// TIA Portal V17 export
// export: Created 2024-08-07T21:44:10.1007869Z, ExportSetting WithDefaults, DisplayName Totally Integrated Automation Portal, DisplayVersion V17 Update 7, DisplayName TIA Portal Openness, DisplayVersion V17 Update 7, DisplayName TIA Portal Version Control Interface, DisplayVersion V17, DisplayName SINAMICS Startdrive Advanced, DisplayVersion V17 SP2, DisplayName SINAMICS Startdrive G110M, G120, G120C, G120D, G120P, G115D, DisplayVersion V17 SP2, DisplayName SINAMICS Startdrive G130, G150, S120, S150, SINAMICS MV, S210, DisplayVersion V17 SP2, DisplayName STEP 7 Professional, DisplayVersion V17 Update 7, DisplayName STEP 7 Safety, DisplayVersion V17 Update 6, DisplayName WinCC Advanced / Unified PC, DisplayVersion V17 Update 7
FUNCTION "FC_DMC" : Void   // FC2012, LAD
{ S7_Optimized_Access := 'TRUE' }
VERSION : 0.1
// stored: AutoNumber false, IsIECCheckEnabled false, SetENOAutomatically false, UDAEnableTagReadback false
   VAR_TEMP
      stationName1 : WString;
      stationName2 : WString;
   END_VAR
BEGIN

REGION Network 1: SET DMC CONNECTION BLOCK
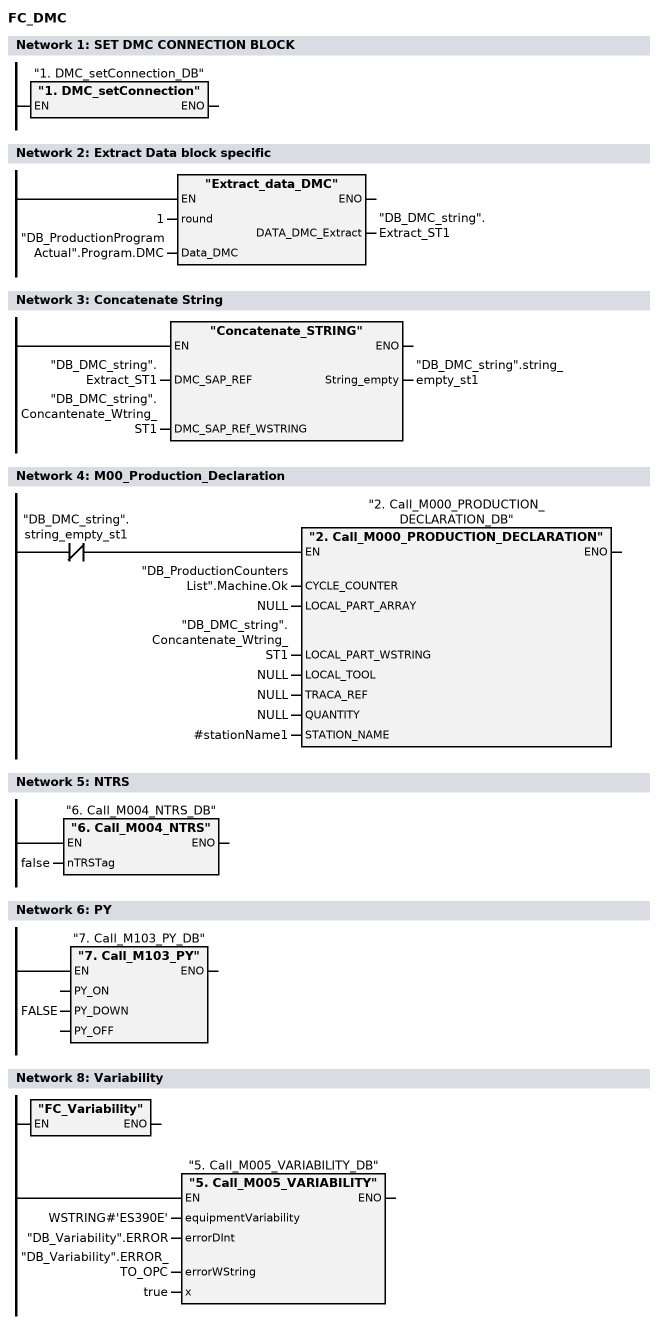
   RUNG wire#powerrail
      "1. DMC_setConnection_DB"()
   END_RUNG
   // the same network as SCL:
   "1. DMC_setConnection_DB"();   // "1. DMC_setConnection"
END_REGION

REGION Network 2: Extract Data block specific
   RUNG wire#powerrail
      "Extract_data_DMC"(round := 1, Data_DMC := "DB_ProductionProgramActual".Program.DMC, DATA_DMC_Extract => "DB_DMC_string".Extract_ST1)
   END_RUNG
   // the same network as SCL:
   "Extract_data_DMC"(round := 1,
                      Data_DMC := "DB_ProductionProgramActual".Program.DMC,
                      DATA_DMC_Extract => "DB_DMC_string".Extract_ST1);
END_REGION

REGION Network 3: Concatenate String
   RUNG wire#powerrail
      "Concatenate_STRING"(DMC_SAP_REF := "DB_DMC_string".Extract_ST1, DMC_SAP_REf_WSTRING := "DB_DMC_string".Concantenate_Wtring_ST1, String_empty => "DB_DMC_string".string_empty_st1)
   END_RUNG
   // the same network as SCL:
   "Concatenate_STRING"(DMC_SAP_REF := "DB_DMC_string".Extract_ST1,
                        DMC_SAP_REf_WSTRING := "DB_DMC_string".Concantenate_Wtring_ST1,
                        String_empty => "DB_DMC_string".string_empty_st1);
END_REGION

REGION Network 4: M00_Production_Declaration
   RUNG wire#powerrail
      I_Contact( "DB_DMC_string".string_empty_st1 )
      "2. Call_M000_PRODUCTION_DECLARATION_DB"(CYCLE_COUNTER := "DB_ProductionCountersList".Machine.Ok, LOCAL_PART_ARRAY := NULL, LOCAL_PART_WSTRING := "DB_DMC_string".Concantenate_Wtring_ST1, LOCAL_TOOL := NULL, TRACA_REF := NULL, QUANTITY := NULL, STATION_NAME := #stationName1)
   END_RUNG
   // the same network as SCL:
   IF NOT "DB_DMC_string".string_empty_st1 THEN
       "2. Call_M000_PRODUCTION_DECLARATION_DB"(CYCLE_COUNTER := "DB_ProductionCountersList".Machine.Ok,   // "2. Call_M000_PRODUCTION_DECLARATION"
                               LOCAL_PART_ARRAY := NULL,
                               LOCAL_PART_WSTRING := "DB_DMC_string".Concantenate_Wtring_ST1,
                               LOCAL_TOOL := NULL,
                               TRACA_REF := NULL,
                               QUANTITY := NULL,
                               STATION_NAME := #stationName1);
   END_IF;
END_REGION

REGION Network 5: NTRS
   RUNG wire#powerrail
      "6. Call_M004_NTRS_DB"(nTRSTag := false)
   END_RUNG
   // the same network as SCL:
   "6. Call_M004_NTRS_DB"(nTRSTag := false);   // "6. Call_M004_NTRS"
END_REGION

REGION Network 6: PY
   RUNG wire#powerrail
      "7. Call_M103_PY_DB"(PY_ON :=, PY_DOWN := FALSE, PY_OFF :=)
   END_RUNG
   // the same network as SCL:
   "7. Call_M103_PY_DB"(PY_DOWN := FALSE);   // "7. Call_M103_PY"
END_REGION

REGION Network 7 (SCL): Icons DMC
   "MII_Parameters".HMI.statusHmiDMC1 := 0;
   "MII_Parameters".HMI.statusHmiDMC2 := 0;
   IF "0. OpcUaClient_DB".connected AND NOT "DB_DMC_string".string_empty_st1 THEN
       "MII_Parameters".HMI.statusHmiDMC1 := 1;
   END_IF;
   IF "0. OpcUaClient_DB".connected AND NOT "DB_DMC_string".string_empty_st2 THEN
       "MII_Parameters".HMI.statusHmiDMC2 := 1;
   END_IF;
END_REGION

REGION Network 8: Variability
   RUNG wire#powerrail
      "FC_Variability"()
   END_RUNG
   RUNG wire#powerrail
      "5. Call_M005_VARIABILITY_DB"(equipmentVariability := WSTRING#'ES390E', errorDInt := "DB_Variability".ERROR, errorWString := "DB_Variability".ERROR_TO_OPC, x := true)
   END_RUNG
   // the same network as SCL:
   "FC_Variability"();
   "5. Call_M005_VARIABILITY_DB"(equipmentVariability := WSTRING#'ES390E',   // "5. Call_M005_VARIABILITY"
                           errorDInt := "DB_Variability".ERROR,
                           errorWString := "DB_Variability".ERROR_TO_OPC,
                           x := true);
END_REGION
END_FUNCTION
